Staubli VAL3: onEdit.pgx

public program onEdit(string& x_sItem[])
  local string l_sItem
  local num l_nValue
  local num l_nValue1
begin
  //
  // compose the string
  // call getType(l_sItem)
  // x_sItem=l_sItem+" ???"
  //
  logMsg("OnEdit")
  call findValue(x_sItem,l_nValue,l_nValue1)
  call use:timerDialog("the value is: "+toString("",l_nValue),2)
end
